// TIA Portal V19 export
TYPE "LEXCHANGETRAY_typeEmActionCostraint"
// stored: Access Published
   STRUCT
      em2 : Bool;
      em3 : Bool;
      em6 : Bool;
   END_STRUCT;
END_TYPE
